ORGANIZATION_BLOCK "CYC_INT5"	// OB 35
TITLE = "Cyclic Interrupt"
VERSION : 0.1
VAR_TEMP
  OB35_EV_CLASS : BYTE ;	//Bits 0-3 = 1 (Coming event), Bits 4-7 = 1 (Event class 1)
  OB35_STRT_INF : BYTE ;	//16#36 (OB 35 has started)
  OB35_PRIORITY : BYTE ;	//Priority of OB Execution
  OB35_OB_NUMBR : BYTE ;	//35 (Organization block 35, OB35)
  OB35_RESERVED_1 : BYTE ;	//Reserved for system
  OB35_RESERVED_2 : BYTE ;	//Reserved for system
  OB35_PHASE_OFFSET : WORD ;	//Phase offset (msec)
  OB35_RESERVED_3 : INT ;	//Reserved for system
  OB35_EXC_FREQ : INT ;	//Frequency of execution (msec)
  OB35_DATE_TIME : DATE_AND_TIME ;	//Date and time OB35 started
  rSetManualPreset_10 : REAL ;
  rKp_10 : REAL ;
  rSetManualPreset_22 : REAL ;
  rKp_22 : REAL ;
  rSetManualPreset_25 : REAL ;
  rKp_25 : REAL ;
  wOut_PQW258 : WORD ;
  wOut_PQW260 : WORD ;
  wOut_PQW262 : WORD ;
  wOut_PQW256 : WORD ;
END_VAR
BEGIN
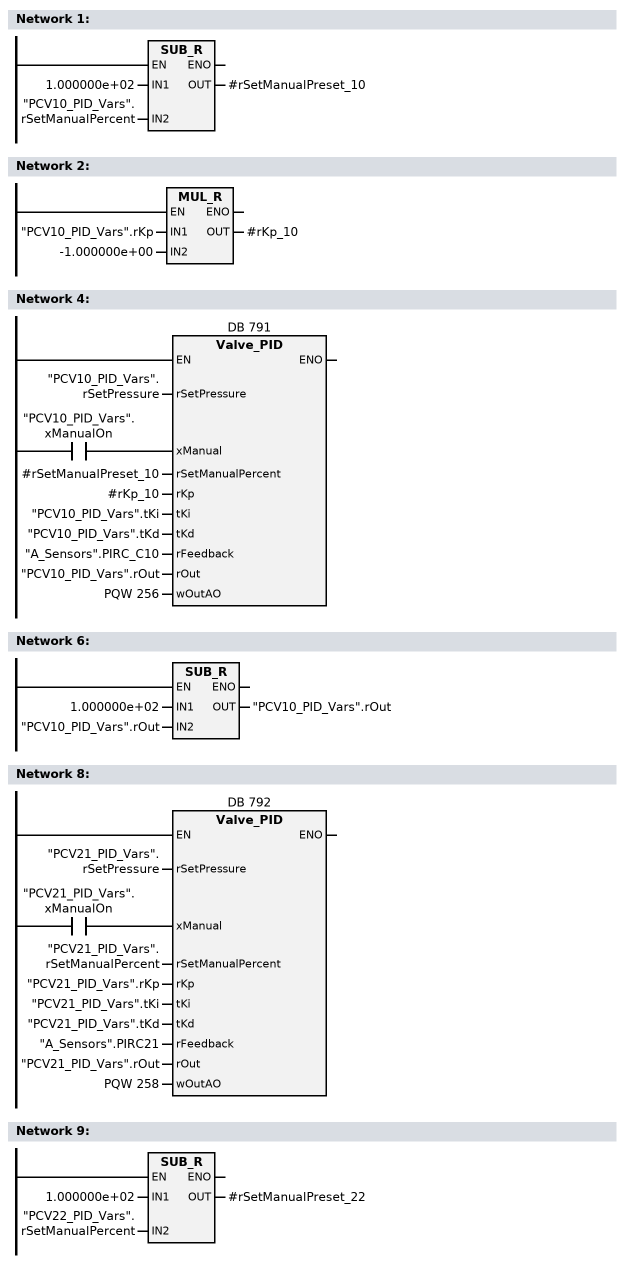
NETWORK
TITLE =
      L     1.000000e+02;
      L     "PCV10_PID_Vars".rSetManualPercent;
      -R;
      T     #rSetManualPreset_10;
      NOP   0;
NETWORK
TITLE =
      L     "PCV10_PID_Vars".rKp;
      L     -1.000000e+00;
      *R;
      T     #rKp_10;
      NOP   0;
NETWORK
TITLE =
NETWORK
TITLE =
      A     "PCV10_PID_Vars".xManualOn;
      =     L 52.0;
      BLD   103;
      CALL  "Valve_PID" , DB 791 (
           rSetPressure             := "PCV10_PID_Vars".rSetPressure,
           xManual                  := L 52.0,
           rSetManualPercent        := #rSetManualPreset_10,
           rKp                      := #rKp_10,
           tKi                      := "PCV10_PID_Vars".tKi,
           tKd                      := "PCV10_PID_Vars".tKd,
           rFeedback                := "A_Sensors".PIRC_C10,
           rOut                     := "PCV10_PID_Vars".rOut,
           wOutAO                   := PQW 256);
      NOP   0;
NETWORK
TITLE =
NETWORK
TITLE =
      L     1.000000e+02;
      L     "PCV10_PID_Vars".rOut;
      -R;
      T     "PCV10_PID_Vars".rOut;
      NOP   0;
NETWORK
TITLE =
NETWORK
TITLE =
      A     "PCV21_PID_Vars".xManualOn;
      =     L 52.0;
      BLD   103;
      CALL  "Valve_PID" , DB 792 (
           rSetPressure             := "PCV21_PID_Vars".rSetPressure,
           xManual                  := L 52.0,
           rSetManualPercent        := "PCV21_PID_Vars".rSetManualPercent,
           rKp                      := "PCV21_PID_Vars".rKp,
           tKi                      := "PCV21_PID_Vars".tKi,
           tKd                      := "PCV21_PID_Vars".tKd,
           rFeedback                := "A_Sensors".PIRC21,
           rOut                     := "PCV21_PID_Vars".rOut,
           wOutAO                   := PQW 258);
      NOP   0;
NETWORK
TITLE =
      L     1.000000e+02;
      L     "PCV22_PID_Vars".rSetManualPercent;
      -R;
      T     #rSetManualPreset_22;
      NOP   0;
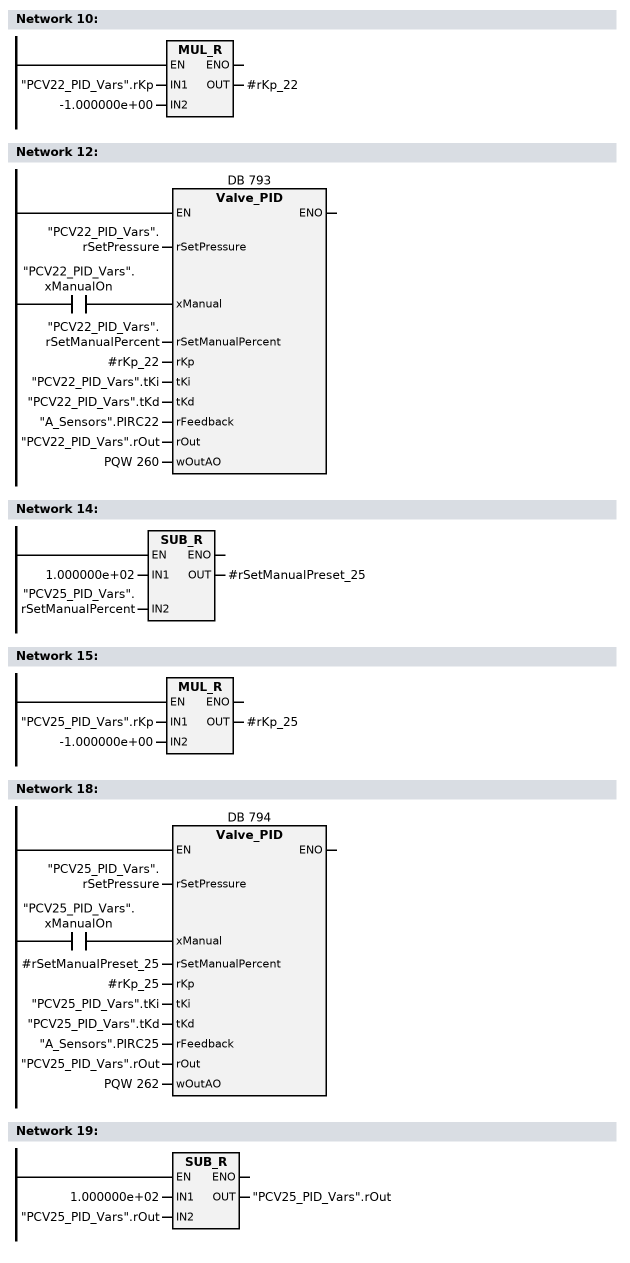
NETWORK
TITLE =
      L     "PCV22_PID_Vars".rKp;
      L     -1.000000e+00;
      *R;
      T     #rKp_22;
      NOP   0;
NETWORK
TITLE =
NETWORK
TITLE =
      A     "PCV22_PID_Vars".xManualOn;
      =     L 52.0;
      BLD   103;
      CALL  "Valve_PID" , DB 793 (
           rSetPressure             := "PCV22_PID_Vars".rSetPressure,
           xManual                  := L 52.0,
           rSetManualPercent        := "PCV22_PID_Vars".rSetManualPercent,
           rKp                      := #rKp_22,
           tKi                      := "PCV22_PID_Vars".tKi,
           tKd                      := "PCV22_PID_Vars".tKd,
           rFeedback                := "A_Sensors".PIRC22,
           rOut                     := "PCV22_PID_Vars".rOut,
           wOutAO                   := PQW 260);
      NOP   0;
NETWORK
TITLE =
NETWORK
TITLE =
      L     1.000000e+02;
      L     "PCV25_PID_Vars".rSetManualPercent;
      -R;
      T     #rSetManualPreset_25;
      NOP   0;
NETWORK
TITLE =
      L     "PCV25_PID_Vars".rKp;
      L     -1.000000e+00;
      *R;
      T     #rKp_25;
      NOP   0;
NETWORK
TITLE =
NETWORK
TITLE =
NETWORK
TITLE =
      A     "PCV25_PID_Vars".xManualOn;
      =     L 52.0;
      BLD   103;
      CALL  "Valve_PID" , DB 794 (
           rSetPressure             := "PCV25_PID_Vars".rSetPressure,
           xManual                  := L 52.0,
           rSetManualPercent        := #rSetManualPreset_25,
           rKp                      := #rKp_25,
           tKi                      := "PCV25_PID_Vars".tKi,
           tKd                      := "PCV25_PID_Vars".tKd,
           rFeedback                := "A_Sensors".PIRC25,
           rOut                     := "PCV25_PID_Vars".rOut,
           wOutAO                   := PQW 262);
      NOP   0;
NETWORK
TITLE =
      L     1.000000e+02;
      L     "PCV25_PID_Vars".rOut;
      -R;
      T     "PCV25_PID_Vars".rOut;
      NOP   0;
END_ORGANIZATION_BLOCK
